FUNCTION_BLOCK ABSTRACT ErrorManagerBase IMPLEMENTS IService
VAR_INPUT
END_VAR
VAR_OUTPUT
END_VAR
VAR
END_VAR

METHOD ABSTRACT AddMessage : BOOL
VAR_INPUT
	i_alarmId: UINT;
	i_active: BOOL;
	//i_acknowledged: BOOL;
	//i_confirmed: BOOL;
	i_severity: ESeverity;
	//i_retain: BOOL;
	i_instanceName: STRING;
END_VAR
END_METHOD

END_FUNCTION_BLOCK

(* stored: Version 1.1.0.1, ProductVersion 3.1.4024.9
   POU ErrorManagerBase: Id {1c21bca8-5546-47f5-85ed-9be3b2000491}, SpecialFunc None
   Method AddMessage: Id {dbea8029-fd7b-46e4-99ce-63c5985aac65} *)
